TYPE IShortTest : 
STRUCT
	bStart :BOOL; //
	bDone  :BOOL; //

   iResult:INT; // 1 OK  2 NG
    
   ErrorID :INT;
   
	

END_STRUCT
END_TYPE

(* stored: Version 1.1.0.1, ProductVersion 3.1.4024.9
   DUT IShortTest: Id {5dc57f6e-0f92-4696-b5e1-0759d407d6e0} *)
